{attribute 'qualified_only'}
// I/O Inputs
//
VAR_GLOBAL

	// Input signals...
	i_HtrTemp AT %I*: REAL; // Heater temperature [°C]
 
END_VAR

(* stored: Version 1.1.0.1, ProductVersion 3.1.4022.6
   GVL IO_Inputs: Id {2a74df3a-f36d-4469-91e6-b72d2d193216} *)
